// LS Electric XG5000 project: 초기화
// PLC NewPLC
// module base 0 slot 0: 입출력 모듈:XBM-DN32H (DC 24V입력/TR 출력, 32점)

PROGRAM NewProgram (task: 스캔 프로그램)

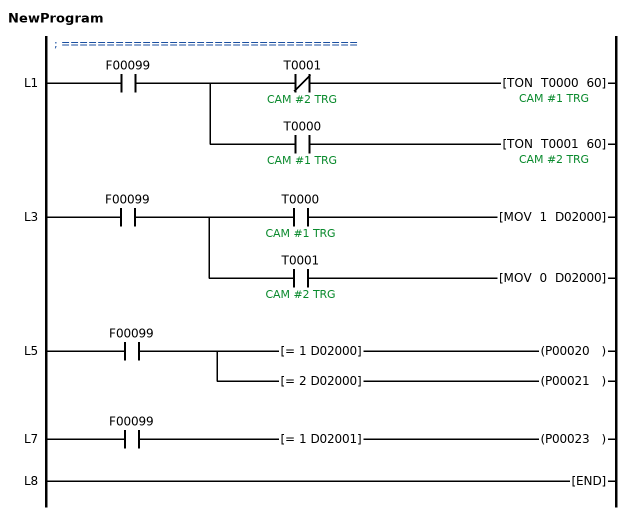
// =================================
; L1
LOAD      F00099
MPUSH
AND NOT   T0001	// CAM #2 TRG
TON       T0000 60	// CAM #1 TRG
MPOP
AND       T0000	// CAM #1 TRG
TON       T0001 60	// CAM #2 TRG
; L3
LOAD      F00099
MPUSH
AND       T0000	// CAM #1 TRG
MOV       1 D02000
MPOP
AND       T0001	// CAM #2 TRG
MOV       0 D02000
; L5
LOAD      F00099
MPUSH
AND=      1 D02000
OUT       P00020
MPOP
AND=      2 D02000
OUT       P00021
; L7
LOAD      F00099
AND=      1 D02001
OUT       P00023
; L8
END

VARIABLES AND COMMENTS (devices not used above)
D02000.0	BIT	CAM #1 TRG
D02000.1	BIT	CAM #2 TRG